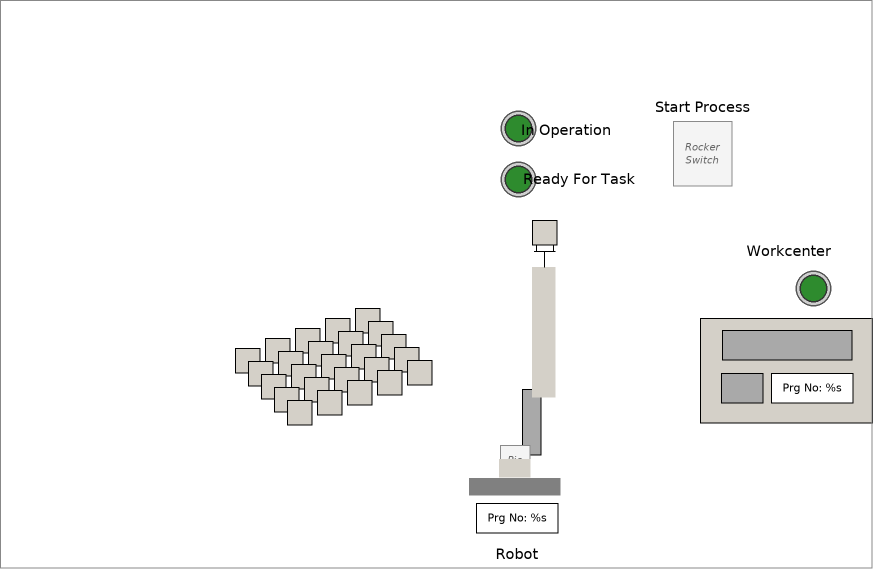
VISUALIZATION Visualization  // 873x569
    RoundedRectangle (522,389 19x66), angle 31, colour toggle: MAIN.RobotWorkcenterControl.RobotPrgNo>0
    RoundedRectangle (355,308 25x25), colour toggle: MAIN.RobotWorkcenterControl.ItemsTable[1,5].Done=TRUE, invisible if: MAIN.RobotWorkcenterControl.ItemsTable[1,5].InProcess=TRUE AND MAIN.RobotWorkcenterControl.ItemsTable[1,5].Done=FALSE
    RoundedRectangle (368,321 25x25), colour toggle: MAIN.RobotWorkcenterControl.ItemsTable[2,5].Done=TRUE, invisible if: MAIN.RobotWorkcenterControl.ItemsTable[2,5].InProcess=TRUE AND MAIN.RobotWorkcenterControl.ItemsTable[2,5].Done=FALSE
    RoundedRectangle (381,334 25x25), colour toggle: MAIN.RobotWorkcenterControl.ItemsTable[3,5].Done=TRUE, invisible if: MAIN.RobotWorkcenterControl.ItemsTable[3,5].InProcess=TRUE AND MAIN.RobotWorkcenterControl.ItemsTable[3,5].Done=FALSE
    RoundedRectangle (394,347 25x25), colour toggle: MAIN.RobotWorkcenterControl.ItemsTable[4,5].Done=TRUE, invisible if: MAIN.RobotWorkcenterControl.ItemsTable[4,5].InProcess=TRUE AND MAIN.RobotWorkcenterControl.ItemsTable[4,5].Done=FALSE
    RoundedRectangle (407,360 25x25), colour toggle: MAIN.RobotWorkcenterControl.ItemsTable[5,5].Done=TRUE, invisible if: MAIN.RobotWorkcenterControl.ItemsTable[5,5].InProcess=TRUE AND MAIN.RobotWorkcenterControl.ItemsTable[5,5].Done=FALSE
    RoundedRectangle (325,318 25x25), colour toggle: MAIN.RobotWorkcenterControl.ItemsTable[1,4].Done=TRUE, invisible if: MAIN.RobotWorkcenterControl.ItemsTable[1,4].InProcess=TRUE AND MAIN.RobotWorkcenterControl.ItemsTable[1,4].Done=FALSE
    RoundedRectangle (338,331 25x25), colour toggle: MAIN.RobotWorkcenterControl.ItemsTable[2,4].Done=TRUE, invisible if: MAIN.RobotWorkcenterControl.ItemsTable[2,4].InProcess=TRUE AND MAIN.RobotWorkcenterControl.ItemsTable[2,4].Done=FALSE
    RoundedRectangle (351,344 25x25), colour toggle: MAIN.RobotWorkcenterControl.ItemsTable[3,4].Done=TRUE, invisible if: MAIN.RobotWorkcenterControl.ItemsTable[3,4].InProcess=TRUE AND MAIN.RobotWorkcenterControl.ItemsTable[3,4].Done=FALSE
    RoundedRectangle (364,357 25x25), colour toggle: MAIN.RobotWorkcenterControl.ItemsTable[4,4].Done=TRUE, invisible if: MAIN.RobotWorkcenterControl.ItemsTable[4,4].InProcess=TRUE AND MAIN.RobotWorkcenterControl.ItemsTable[4,4].Done=FALSE
    RoundedRectangle (377,370 25x25), colour toggle: MAIN.RobotWorkcenterControl.ItemsTable[5,4].Done=TRUE, invisible if: MAIN.RobotWorkcenterControl.ItemsTable[5,4].InProcess=TRUE AND MAIN.RobotWorkcenterControl.ItemsTable[5,4].Done=FALSE
    RoundedRectangle (295,328 25x25), colour toggle: MAIN.RobotWorkcenterControl.ItemsTable[1,3].Done=TRUE, invisible if: MAIN.RobotWorkcenterControl.ItemsTable[1,3].InProcess=TRUE AND MAIN.RobotWorkcenterControl.ItemsTable[1,3].Done=FALSE
    RoundedRectangle (308,341 25x25), colour toggle: MAIN.RobotWorkcenterControl.ItemsTable[2,3].Done=TRUE, invisible if: MAIN.RobotWorkcenterControl.ItemsTable[2,3].InProcess=TRUE AND MAIN.RobotWorkcenterControl.ItemsTable[2,3].Done=FALSE
    RoundedRectangle (321,354 25x25), colour toggle: MAIN.RobotWorkcenterControl.ItemsTable[3,3].Done=TRUE, invisible if: MAIN.RobotWorkcenterControl.ItemsTable[3,3].InProcess=TRUE AND MAIN.RobotWorkcenterControl.ItemsTable[3,3].Done=FALSE
    RoundedRectangle (334,367 25x25), colour toggle: MAIN.RobotWorkcenterControl.ItemsTable[4,3].Done=TRUE, invisible if: MAIN.RobotWorkcenterControl.ItemsTable[4,3].InProcess=TRUE AND MAIN.RobotWorkcenterControl.ItemsTable[4,3].Done=FALSE
    RoundedRectangle (347,380 25x25), colour toggle: MAIN.RobotWorkcenterControl.ItemsTable[5,3].Done=TRUE, invisible if: MAIN.RobotWorkcenterControl.ItemsTable[5,3].InProcess=TRUE AND MAIN.RobotWorkcenterControl.ItemsTable[5,3].Done=FALSE
    RoundedRectangle (265,338 25x25), colour toggle: MAIN.RobotWorkcenterControl.ItemsTable[1,2].Done=TRUE, invisible if: MAIN.RobotWorkcenterControl.ItemsTable[1,2].InProcess=TRUE AND MAIN.RobotWorkcenterControl.ItemsTable[1,2].Done=FALSE
    RoundedRectangle (278,351 25x25), colour toggle: MAIN.RobotWorkcenterControl.ItemsTable[2,2].Done=TRUE, invisible if: MAIN.RobotWorkcenterControl.ItemsTable[2,2].InProcess=TRUE AND MAIN.RobotWorkcenterControl.ItemsTable[2,2].Done=FALSE
    RoundedRectangle (291,364 25x25), colour toggle: MAIN.RobotWorkcenterControl.ItemsTable[3,2].Done=TRUE, invisible if: MAIN.RobotWorkcenterControl.ItemsTable[3,2].InProcess=TRUE AND MAIN.RobotWorkcenterControl.ItemsTable[3,2].Done=FALSE
    RoundedRectangle (304,377 25x25), colour toggle: MAIN.RobotWorkcenterControl.ItemsTable[4,2].Done=TRUE, invisible if: MAIN.RobotWorkcenterControl.ItemsTable[4,2].InProcess=TRUE AND MAIN.RobotWorkcenterControl.ItemsTable[4,2].Done=FALSE
    RoundedRectangle (317,390 25x25), colour toggle: MAIN.RobotWorkcenterControl.ItemsTable[5,2].Done=TRUE, invisible if: MAIN.RobotWorkcenterControl.ItemsTable[5,2].InProcess=TRUE AND MAIN.RobotWorkcenterControl.ItemsTable[5,2].Done=FALSE
    RoundedRectangle (235,348 25x25), colour toggle: MAIN.RobotWorkcenterControl.ItemsTable[1,1].Done=TRUE, invisible if: MAIN.RobotWorkcenterControl.ItemsTable[1,1].InProcess=TRUE AND MAIN.RobotWorkcenterControl.ItemsTable[1,1].Done=FALSE
    RoundedRectangle (248,361 25x25), colour toggle: MAIN.RobotWorkcenterControl.ItemsTable[2,1].Done=TRUE, invisible if: MAIN.RobotWorkcenterControl.ItemsTable[2,1].InProcess=TRUE AND MAIN.RobotWorkcenterControl.ItemsTable[2,1].Done=FALSE
    RoundedRectangle (261,374 25x25), colour toggle: MAIN.RobotWorkcenterControl.ItemsTable[3,1].Done=TRUE, invisible if: MAIN.RobotWorkcenterControl.ItemsTable[3,1].InProcess=TRUE AND MAIN.RobotWorkcenterControl.ItemsTable[3,1].Done=FALSE
    RoundedRectangle (274,387 25x25), colour toggle: MAIN.RobotWorkcenterControl.ItemsTable[4,1].Done=TRUE, invisible if: MAIN.RobotWorkcenterControl.ItemsTable[4,1].InProcess=TRUE AND MAIN.RobotWorkcenterControl.ItemsTable[4,1].Done=FALSE
    RoundedRectangle (287,400 25x25), colour toggle: MAIN.RobotWorkcenterControl.ItemsTable[5,1].Done=TRUE, invisible if: MAIN.RobotWorkcenterControl.ItemsTable[5,1].InProcess=TRUE AND MAIN.RobotWorkcenterControl.ItemsTable[5,1].Done=FALSE
    Lamp1 (478,108 81x41), variable: MAIN.RobotWorkcenterControl.InOperation, style: Lamp-Lamp1-Green
    Lamp1 (772,268 83x41), variable: MAIN.RobotWorkcenterControl.WorkcenterPrgNo > 0, style: Lamp-Lamp1-Green
    Rectangle (700,318 173x105), colour toggle: MAIN.RobotWorkcenterControl.WorkcenterPrgNo > 0
    RoundedRectangle (722,330 130x30), colour toggle: MAIN.RobotWorkcenterControl.WorkcenterPrgNo > 0
    RoundedRectangle (721,373 42x30), colour toggle: MAIN.RobotWorkcenterControl.WorkcenterPrgNo > 0
    RoundedRectangle (771,373 82x30), "Prg No: %s", text variable: MAIN.RobotWorkcenterControl.WorkcenterPrgNo
    RockerSwitch (673,121 59x65), variable: MAIN.Start, behaviour: TOGGLE, style: Switch-RockerSwitch-Gray
    Label (648,92 109x30), "Start Process"
    Label (741,236 96x30), "Workcenter"
    Lamp1 (478,159 81x41), variable: MAIN.RobotWorkcenterControl.ReadyForNewTask, style: Lamp-Lamp1-Green
    Label (518,115 109x30), "In Operation"
    Label (520,164 123x30), "Ready For Task"
    Rectangle (469,478 91x17)
    Pie (500,445 30x30)
    Rectangle (499,459 31x18)
    Rectangle (532,267 23x130), colour toggle: MAIN.RobotWorkcenterControl.RobotPrgNo>0
        p2858320360: MAIN.RobotSimulation.ArmPosition
    RoundedRectangle (476,503 82x30), "Prg No: %s", text variable: MAIN.RobotWorkcenterControl.RobotPrgNo
    Label (469,539 96x30), "Robot"
    Line (544,251) (544,267)
        p2858320360: MAIN.RobotSimulation.ArmPosition
    Line (534,251) (555,251)
        p2858320360: MAIN.RobotSimulation.ArmPosition
    Line (536,233) (536,251)
        p2858320360: MAIN.RobotSimulation.ArmPosition
    Line (553,233) (553,251)
        p2858320360: MAIN.RobotSimulation.ArmPosition
    RoundedRectangle (532,220 25x25), colour toggle: MAIN.RobotWorkcenterControl.RobotPrgNo=2, invisible if: MAIN.RobotWorkcenterControl.RobotPrgNo<=0
        p2858320360: MAIN.RobotSimulation.ArmPosition
END_VISUALIZATION

(* stored: Version 1.1.0.1, ProductVersion 3.1.4024.15
   Visu Visualization: Id {f779ea86-b836-4542-912f-ccfcc493618b} *)
